{attribute 'qualified_only'}
VAR_GLOBAL
	StartCommand1		: StartCommand;
	AddCommand1			: AddCommand 			:= (Val1 := 3, Val2 := 2);
	DelayedAddCommand1	: DelayedAddCommand 	:= (Val1 := 4, Val2 := 5);
END_VAR

(* stored: Version 1.1.0.1, ProductVersion 3.1.4022.10
   GVL Commands: Id {6236b5d6-4821-0594-19ad-760d9d192eb5} *)
